FUNCTION_BLOCK AGENT_SEND (* Sends diagnostic data to the remote agent *)
  (* Standard: 61499-2; Type: Service Interface Function Block; Description: This function block type manages a TCP/IP client connection to a remote diagnostic agent server. For each  input event it receives, data is sent as a packet to the server. Configuration parameters for the server address, server listener port and data type allow each function block instance to create their own data channel for use during the diagnostic session. *)
  (* Version 1.0, 2019-01-09, badger *)
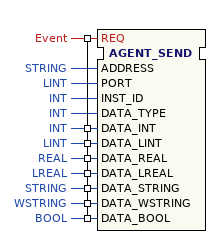
  EVENT_INPUT
    REQ WITH DATA_INT, DATA_LINT, DATA_LREAL, DATA_STRING, DATA_BOOL, DATA_REAL, DATA_WSTRING; (* Service Request *)
  END_EVENT
  VAR_INPUT
    ADDRESS : STRING; (* Address of the remote diagnostic server. *)
    PORT : LINT; (* Port on the remote diagnostic server to connect to. *)
    INST_ID : INT; (* Function block instance ID *)
    DATA_TYPE : INT; (* Enumerated data type of the input currently being watched. *)
    DATA_INT : INT; (* Integer data input *)
    DATA_LINT : LINT; (* Long integer data input *)
    DATA_REAL : REAL; (* Data type Real *)
    DATA_LREAL : LREAL; (* Long Real number (used with double or float data types) *)
    DATA_STRING : STRING; (* String data type *)
    DATA_WSTRING : WSTRING; (* Wide String data type *)
    DATA_BOOL : BOOL; (* Boolean data type *)
  END_VAR
  SERVICE APPLICATION/RESOURCE (* Sends diagnostic data to the remote agent *)
    SEQUENCE normal_establishment
      APPLICATION.INIT+(PARAMS) -> RESOURCE.initialize(PARAMS) -> APPLICATION.INITO+();
    END_SEQUENCE
    SEQUENCE unsuccessful_establishment
      APPLICATION.INIT+(PARAMS) -> RESOURCE.initialize(PARAMS) -> APPLICATION.INITO-(STATUS);
    END_SEQUENCE
    SEQUENCE request_confirm
      APPLICATION.REQ+(SD) -> RESOURCE.request(SD) -> APPLICATION.CNF+(RD);
    END_SEQUENCE
    SEQUENCE request_inhibited
      APPLICATION.REQ-(SD) -> APPLICATION.CNF-(STATUS);
    END_SEQUENCE
    SEQUENCE request_error
      APPLICATION.REQ+(SD) -> RESOURCE.request(SD) -> APPLICATION.CNF-(STATUS);
    END_SEQUENCE
    SEQUENCE indication_response
      RESOURCE.indicate(RD) -> APPLICATION.IND+(RD);
      APPLICATION.RSP(QI,SD) -> RESOURCE.response(QI,SD);
    END_SEQUENCE
    SEQUENCE indication_inhibited
      RESOURCE.indicate(RD,QI=FALSE) -> RESOURCE.inhibited();
    END_SEQUENCE
    SEQUENCE error_indication
      RESOURCE.error(STATUS) -> APPLICATION.IND-(STATUS);
    END_SEQUENCE
    SEQUENCE application_initiated_termination
      APPLICATION.INIT-() -> RESOURCE.terminate() -> APPLICATION.INITO-(STATUS);
    END_SEQUENCE
    SEQUENCE resource_initiated_termination
      -> APPLICATION.INITO-(STATUS);
    END_SEQUENCE
  END_SERVICE
END_FUNCTION_BLOCK
